(* PLC project SafeLOGIC, BrAutomation SafeDESIGNER  5.24.1.0 *)
(* stored: companyURL http://www.br-automation.com, creationDateTime Fri Nov 28 15:25:49 2025 *)

PROGRAM DI_MON_PARA
  VAR  (* added by the conversion: wires and edge detectors of the diagram *)
    _NOT_S18_OUT : ANY;
  END_VAR

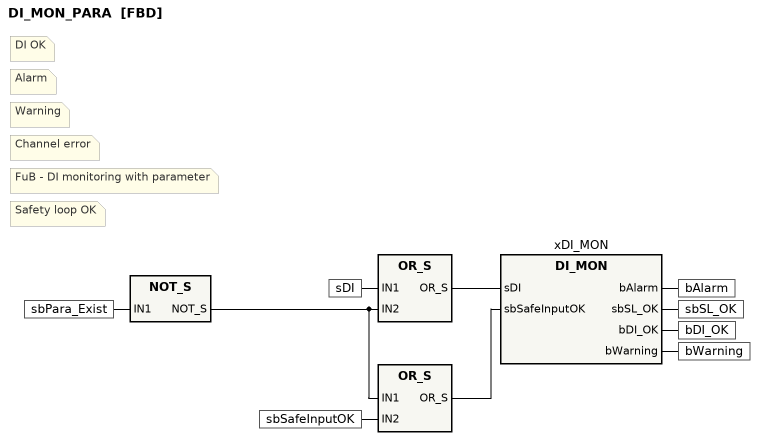
(* FBD diagram, written out as Structured Text *)
(* FuB - DI monitoring with parameter *)
(* Alarm *)
(* Safety loop OK *)
(* DI OK *)
(* Channel error *)
(* Warning *)
_NOT_S18_OUT := NOT_S(sbPara_Exist);
xDI_MON(sDI := OR_S(sDI, _NOT_S18_OUT), sbSafeInputOK := OR_S(_NOT_S18_OUT, sbSafeInputOK));
bWarning := xDI_MON.bWarning;
bDI_OK := xDI_MON.bDI_OK;
sbSL_OK := xDI_MON.sbSL_OK;
bAlarm := xDI_MON.bAlarm;
END_PROGRAM
